// TIA Portal project "Poka Yoke Directa_V18" (V18)

(* hardware
DEVICE "S7-1200 station_1"  S7-1200 Station
   slot 0: "Rack_0"  S7-1200 Rack  Rack  V1.0
   slot 1: "PLC_1"  CPU 1215C DC/DC/Rly  6ES7 215-1HG40-0XB0  V4.6
DEVICE "GSD device_1"  GSD.Device.PN
   slot 0: "Rack"  Rack  V1.0
   slot 0: "smart-runner"  SmartRunner  310754  V3.1
      slot 0: "SmartRunner"  SmartRunner
      slot 1: "PN Interface"  PN Interface
         slot 1: "Port 1"  Port 1
         slot 2: "Port 2"  Port 2
   slot 1: "Head Address 1_1"  Head Address 1
      slot 0: "Head Address 1"  Head Address 1
*)

// ===== PLC "PLC_1"  CPU 1215C DC/DC/Rly =====

VAR_GLOBAL   // PLC tag table "PLC"
   "Pulsador Rojo Reset Desvio" AT %I0.0 : Bool;
   "No Match - RS482" AT %I0.1 : Bool;   // Sensor 2 - Mediante R482
   "Sensor Inductivo Soporte" AT %I0.2 : Bool;
   "Error" AT %I68.0 : Bool;
   "No Match - Profinet" AT %I68.1 : Bool;   // Sensor 1 - Profinet
   "Warning" AT %I68.2 : Bool;
   "Event" AT %I68.3 : Bool;
   "Status_addr" AT %I68.4 : Bool;
   "Status_addr 1" AT %I68.5 : Bool;
   "Result" AT %IB69 : Byte;
   "Counter" AT %IB70 : Byte;
   "Quality A" AT %IB71 : Byte;
   "Quality B" AT %IB72 : Byte;
   "Quality C" AT %IB73 : Byte;
   "Pos X" AT %IW74 : Int;
   "Pos Z" AT %IW76 : Int;
   "Checksum" AT %IB78 : Byte;
   "Rele Baliza" AT %Q0.3 : Bool;
   "Piloto Pulsador Rojo" AT %Q0.0 : Bool;
   "Rele bocina intermitente" AT %Q0.1 : Bool;
   "Trigger" AT %Q69.0 : Bool;
   "Teach" AT %Q71.0 : Bool;
   "Choose Profile" AT %QB73 : Byte;
   "Parada Gantry" AT %Q0.4 : Bool;
   "Piloto Error CPU" AT %Q0.5 : Bool;
   "Piloto OK" AT %Q0.2 : Bool;
   "Flanco Sensor Inductivo" AT %M0.2 : Bool;
   "Resultante" AT %MW10 : Int;
   "PF_Profinet" AT %MW2 : Hw_Io;
   "PF_LED" AT %MW4 : UInt;
   "System_Byte" AT %MB500 : Byte;
   "FirstScan" AT %M500.0 : Bool;
   "DiagStatusUpdate" AT %M500.1 : Bool;
   "AlwaysTRUE" AT %M500.2 : Bool;
   "AlwaysFALSE" AT %M500.3 : Bool;
   "Prueba" AT %M0.0 : Bool;
END_VAR

DATA_BLOCK "DataLogger_DB"   // DB9
{ S7_Optimized_Access := 'TRUE' }
VERSION : 0.1
// stored: InstanceOfName DataLogger
"DataLogger"
BEGIN
END_DATA_BLOCK

DATA_BLOCK "Control DataLogger"   // DB10
{ S7_Optimized_Access := 'TRUE' }
VERSION : 0.1
   VAR
      "Abrir Archivo" : Bool;
      "Escribir Archivo" : Bool;
      "Crear Archivo" : Bool;
      "Cerrar Archivo" : Bool;
      ID : DWord := 16#20;
   END_VAR
   VAR RETAIN
      "Name" : String;
   END_VAR
   VAR
      Data : Struct
         "Sensor 1" : Bool;
         "Sensor 2" : Bool;
         "Conexion Profinet" : Bool;
         "Quality A" : Int;
         "Quality B" : Int;
         "Quality C" : Int;
      END_STRUCT;
   END_VAR
BEGIN
END_DATA_BLOCK

// folder: 10_Sensor Doble

DATA_BLOCK "Status_LED"   // DB13
{ S7_Optimized_Access := 'TRUE' }
VERSION : 0.1
   VAR
      HW : Hw_Io := 50;
      LED : UInt := 2;
      "Return" : Int;
   END_VAR
BEGIN
END_DATA_BLOCK

// folder: FBs

DATA_BLOCK "SmartRunnner_Control_DB"   // DB8
{ S7_Optimized_Access := 'TRUE' }
VERSION : 0.1
// stored: InstanceOfName SmartRunnner_Control
"SmartRunnner_Control"
BEGIN
END_DATA_BLOCK

// folder: System blocks/Program resources

DATA_BLOCK "Temporizador TON Lectura de Datos"   // DB1
{ S7_Optimized_Access := 'TRUE' }
AUTHOR : Simatic
FAMILY : IEC
NAME : IEC_TMR
VERSION : 1.0
// stored: InstanceOfName IEC_TIMER
"IEC_TIMER"
BEGIN
END_DATA_BLOCK

DATA_BLOCK "Temporizador TON Pulsador Rojo"   // DB2
{ S7_Optimized_Access := 'TRUE' }
AUTHOR : Simatic
FAMILY : IEC
NAME : IEC_TMR
VERSION : 1.0
// stored: InstanceOfName IEC_TIMER
"IEC_TIMER"
BEGIN
END_DATA_BLOCK

DATA_BLOCK "Temporizador TP Pulsador Rojo"   // DB3
{ S7_Optimized_Access := 'TRUE' }
AUTHOR : Simatic
FAMILY : IEC
NAME : IEC_TMR
VERSION : 1.0
// stored: InstanceOfName IEC_TIMER
"IEC_TIMER"
BEGIN
END_DATA_BLOCK

DATA_BLOCK "Temporizador TP Reset"   // DB4
{ S7_Optimized_Access := 'TRUE' }
AUTHOR : Simatic
FAMILY : IEC
NAME : IEC_TMR
VERSION : 1.0
// stored: InstanceOfName IEC_TIMER
"IEC_TIMER"
BEGIN
END_DATA_BLOCK

DATA_BLOCK "Temporizador TON Reset"   // DB5
{ S7_Optimized_Access := 'TRUE' }
AUTHOR : Simatic
FAMILY : IEC
NAME : IEC_TMR
VERSION : 1.0
// stored: InstanceOfName IEC_TIMER
"IEC_TIMER"
BEGIN
END_DATA_BLOCK

DATA_BLOCK "TON_BOCINA"   // DB6
{ S7_Optimized_Access := 'TRUE' }
AUTHOR : Simatic
FAMILY : IEC
NAME : IEC_TMR
VERSION : 1.0
// stored: InstanceOfName IEC_TIMER
"IEC_TIMER"
BEGIN
END_DATA_BLOCK

DATA_BLOCK "TP_BOCINA"   // DB7
{ S7_Optimized_Access := 'TRUE' }
AUTHOR : Simatic
FAMILY : IEC
NAME : IEC_TMR
VERSION : 1.0
// stored: InstanceOfName IEC_TIMER
"IEC_TIMER"
BEGIN
END_DATA_BLOCK

DATA_BLOCK "TP Guardado"   // DB11
{ S7_Optimized_Access := 'TRUE' }
AUTHOR : Simatic
FAMILY : IEC
NAME : IEC_TMR
VERSION : 1.0
// stored: InstanceOfName IEC_TIMER
"IEC_TIMER"
BEGIN
END_DATA_BLOCK

DATA_BLOCK "Temporizador TON Giro Pieza"   // DB12
{ S7_Optimized_Access := 'TRUE' }
AUTHOR : Simatic
FAMILY : IEC
NAME : IEC_TMR
VERSION : 1.0
// stored: InstanceOfName IEC_TIMER
"IEC_TIMER"
BEGIN
END_DATA_BLOCK

DATA_BLOCK "TON Guardado"   // DB14
{ S7_Optimized_Access := 'TRUE' }
AUTHOR : Simatic
FAMILY : IEC
NAME : IEC_TMR
VERSION : 1.0
// stored: InstanceOfName IEC_TIMER
"IEC_TIMER"
BEGIN
END_DATA_BLOCK

DATA_BLOCK "Temporizador TP Lectura de Datos"   // DB25
{ S7_Optimized_Access := 'TRUE' }
AUTHOR : Simatic
FAMILY : IEC
NAME : IEC_TMR
VERSION : 1.0
// stored: InstanceOfName IEC_TIMER
"IEC_TIMER"
BEGIN
END_DATA_BLOCK

// folder: (top level)

FUNCTION_BLOCK "DataLogger"   // FB2, LAD
{ S7_Optimized_Access := 'TRUE' }
VERSION : 0.1
   VAR_INPUT
      LogCreate : Bool;
      LogOpen : Bool;
      LogWrite : Bool;
      LogClose : Bool;
      "Name" : String := 'Datalogger';
   END_VAR
   VAR_IN_OUT
      Data : Struct
         RS482 : Bool;
         Profinet : Bool;
         "Conexion Profinet" : Bool;
         "Quality A" : Int;
         "Quality B" : Int;
         "Quality C" : Int;
      END_STRUCT;
      ID : DWord := 16#20;
   END_VAR
   VAR
      Create : DataLogCreate;
      Header : String := 'RS482,Profinet,Conexion Profinet,Quality A, Quality B, Quality C';
      CreateDone : Bool;
      Write : DataLogWrite;
      WriteDone : Bool;
      OpenDone : Bool;
      Open : DataLogOpen;
      DataLogClose : DataLogClose;
   END_VAR
   VAR CONSTANT
      Records : UDInt := 20000;
      Format : UInt := 1;
      Timestamp : UInt := 4;
      Mode : UInt := 0;
   END_VAR
BEGIN

REGION Network 1
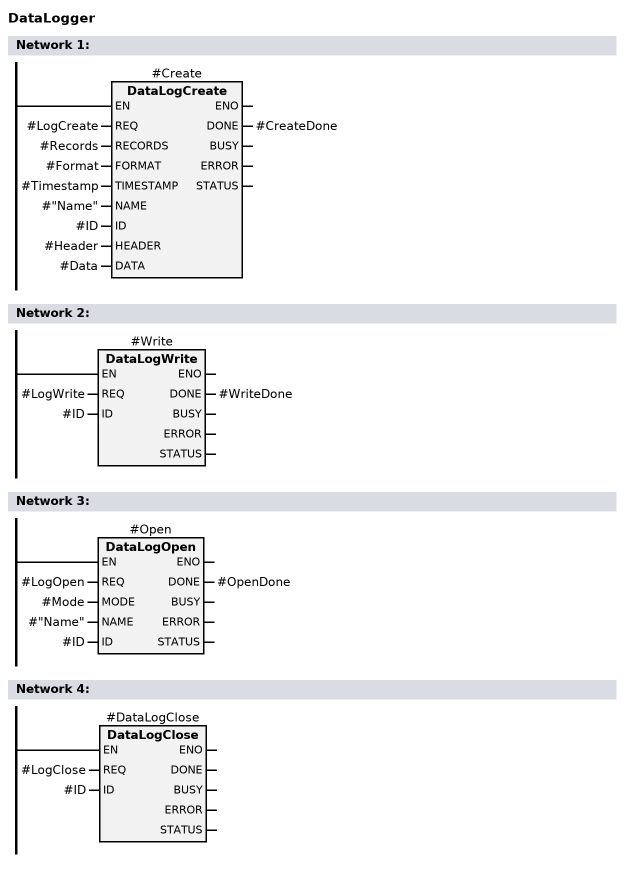
   #Create(REQ := #LogCreate,   // DataLogCreate
           RECORDS := #Records,
           FORMAT := #Format,
           TIMESTAMP := #Timestamp,
           "NAME" := #"Name",
           ID := #ID,
           HEADER := #Header,
           DATA := #Data,
           DONE => #CreateDone);
END_REGION

REGION Network 2
   #Write(REQ := #LogWrite, ID := #ID, DONE => #WriteDone);   // DataLogWrite
END_REGION

REGION Network 3
   #Open(REQ := #LogOpen, MODE := #Mode, "NAME" := #"Name", ID := #ID, DONE => #OpenDone);   // DataLogOpen
END_REGION

REGION Network 4
   #DataLogClose(REQ := #LogClose, ID := #ID);   // DataLogClose
END_REGION
END_FUNCTION_BLOCK

FUNCTION "Conversion Byte a Int" : Void   // FC2, LAD
{ S7_Optimized_Access := 'TRUE' }
VERSION : 0.1
BEGIN

REGION Network 1 (SCL)
   //comentario de prueba
   "Control DataLogger".Data."Quality A" :=  BYTE_TO_INT(IN :="Quality A");
   "Control DataLogger".Data."Quality B" := BYTE_TO_INT(IN := "Quality B");
   "Control DataLogger".Data."Quality C" := BYTE_TO_INT(IN := "Quality C");
END_REGION
END_FUNCTION

ORGANIZATION_BLOCK "Main"   // OB1, LAD, ProgramCycle
TITLE = "Main Program Sweep (Cycle)"
{ S7_Optimized_Access := 'TRUE' }
VERSION : 0.1
   VAR_INPUT
      Initial_Call : Bool;   // Initial call of this OB
      Remanence : Bool;   // =True, if remanent data are available
   END_VAR
BEGIN

REGION Network 1: Lectura del ambos sensores
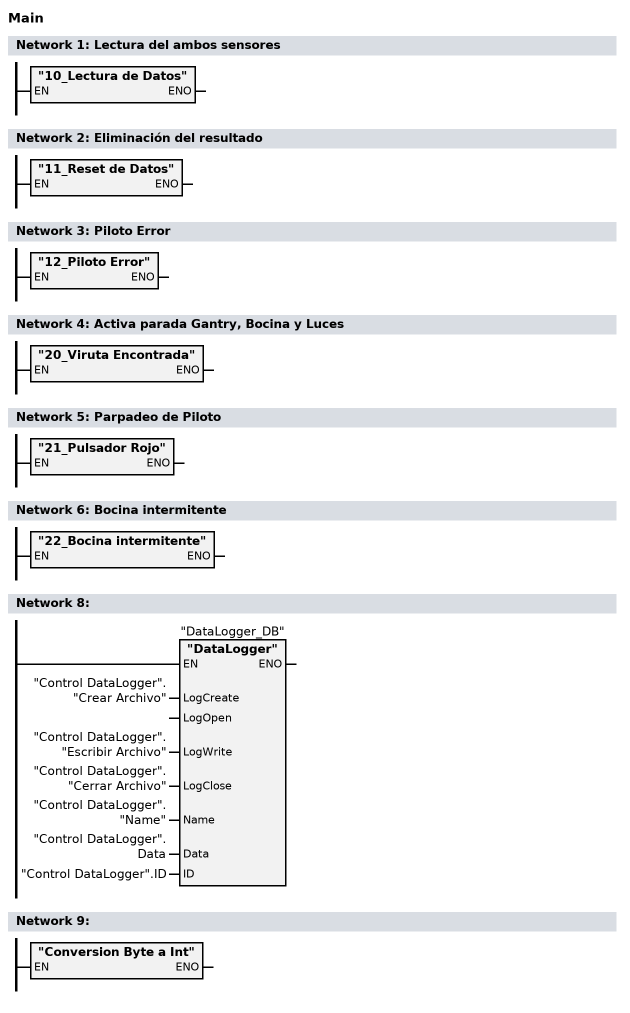
   RUNG wire#powerrail
      "10_Lectura de Datos"()
   END_RUNG
   // the same network as SCL:
   "10_Lectura de Datos"();
END_REGION

REGION Network 2: Eliminación del resultado
   RUNG wire#powerrail
      "11_Reset de Datos"()
   END_RUNG
   // the same network as SCL:
   "11_Reset de Datos"();
END_REGION

REGION Network 3: Piloto Error
   RUNG wire#powerrail
      "12_Piloto Error"()
   END_RUNG
   // the same network as SCL:
   "12_Piloto Error"();
END_REGION

REGION Network 4: Activa parada Gantry, Bocina y Luces
   RUNG wire#powerrail
      "20_Viruta Encontrada"()
   END_RUNG
   // the same network as SCL:
   "20_Viruta Encontrada"();
END_REGION

REGION Network 5: Parpadeo de Piloto
   RUNG wire#powerrail
      "21_Pulsador Rojo"()
   END_RUNG
   // the same network as SCL:
   "21_Pulsador Rojo"();
END_REGION

REGION Network 6: Bocina intermitente
   RUNG wire#powerrail
      "22_Bocina intermitente"()
   END_RUNG
   // the same network as SCL:
   "22_Bocina intermitente"();
END_REGION

REGION Network 7 (SCL)
   "Control DataLogger".Data."Sensor 1" := "No Match - RS482";
   "Control DataLogger".Data."Sensor 2" := "No Match - Profinet";
   "Control DataLogger".Data."Conexion Profinet" := "Piloto Error CPU";
END_REGION

REGION Network 8
   RUNG wire#powerrail
      "DataLogger_DB"(LogCreate := "Control DataLogger"."Crear Archivo", LogOpen :=, LogWrite := "Control DataLogger"."Escribir Archivo", LogClose := "Control DataLogger"."Cerrar Archivo", "Name" := "Control DataLogger"."Name", Data := "Control DataLogger".Data, ID := "Control DataLogger".ID)
   END_RUNG
   // the same network as SCL:
   "DataLogger_DB"(LogCreate := "Control DataLogger"."Crear Archivo",   // "DataLogger"
                   LogWrite := "Control DataLogger"."Escribir Archivo",
                   LogClose := "Control DataLogger"."Cerrar Archivo",
                   "Name" := "Control DataLogger"."Name",
                   Data := "Control DataLogger".Data,
                   ID := "Control DataLogger".ID);
END_REGION

REGION Network 9
   RUNG wire#powerrail
      "Conversion Byte a Int"()
   END_RUNG
   // the same network as SCL:
   "Conversion Byte a Int"();
END_REGION
END_ORGANIZATION_BLOCK

// folder: 10_Sensor Doble

FUNCTION "12_Piloto Error" : Void   // FC1, LAD
{ S7_Optimized_Access := 'TRUE' }
VERSION : 0.1
   VAR_TEMP
      PepperF_profinet : Hw_Io;
   END_VAR
BEGIN

REGION Network 1
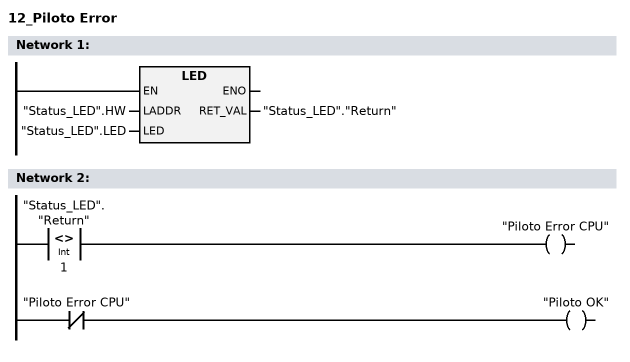
   "Status_LED"."Return" := LED(LADDR := "Status_LED".HW, LED := "Status_LED".LED);
END_REGION

REGION Network 2
   RUNG wire#powerrail
      { S7_Templates := "SrcType := Int" } NE_Contact(in1 := "Status_LED"."Return", in2 := 1)
      Coil( "Piloto Error CPU" )
   END_RUNG
   RUNG wire#powerrail
      I_Contact( "Piloto Error CPU" )
      Coil( "Piloto OK" )
   END_RUNG
   // the same network as SCL:
   "Piloto Error CPU" := "Status_LED"."Return" <> 1;
   "Piloto OK" := NOT "Piloto Error CPU";
END_REGION
END_FUNCTION

FUNCTION "10_Lectura de Datos" : Void   // FC20, LAD
{ S7_Optimized_Access := 'TRUE' }
VERSION : 0.1
   VAR_TEMP   // added for the SCL form of the ladder/FBD networks
      _w1 : Bool;
   END_VAR
BEGIN

REGION Network 1
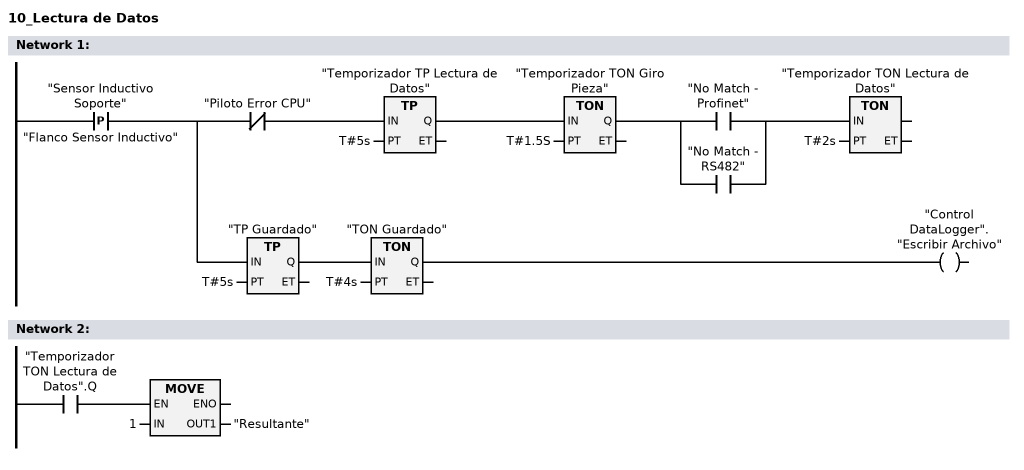
   #_w1 := "Sensor Inductivo Soporte" AND NOT "Flanco Sensor Inductivo";   // rising edge of "Sensor Inductivo Soporte"
   "Flanco Sensor Inductivo" := "Sensor Inductivo Soporte";
   "Temporizador TP Lectura de Datos".TP(IN := #_w1 AND NOT "Piloto Error CPU", PT := T#5s);
   "Temporizador TON Giro Pieza".TON(IN := "Temporizador TP Lectura de Datos".Q, PT := T#1.5S);
   "Temporizador TON Lectura de Datos".TON(IN := "Temporizador TON Giro Pieza".Q AND ("No Match - Profinet" OR "No Match - RS482"),
                           PT := T#2s);
   "TP Guardado".TP(IN := #_w1, PT := T#5s);
   "TON Guardado".TON(IN := "TP Guardado".Q, PT := T#4s);
   "Control DataLogger"."Escribir Archivo" := "TON Guardado".Q;
END_REGION

REGION Network 2
   RUNG wire#powerrail
      Contact( "Temporizador TON Lectura de Datos".Q )
      Move(in := 1, out1 => "Resultante")
   END_RUNG
   // the same network as SCL:
   IF "Temporizador TON Lectura de Datos".Q THEN "Resultante" := 1; END_IF;
END_REGION
END_FUNCTION

FUNCTION "11_Reset de Datos" : Void   // FC21, LAD
{ S7_Optimized_Access := 'TRUE' }
VERSION : 0.1
BEGIN

REGION Network 1
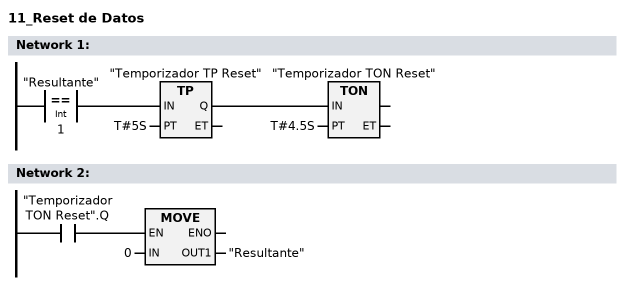
   "Temporizador TP Reset".TP(IN := "Resultante" = 1, PT := T#5S);
   "Temporizador TON Reset".TON(IN := "Temporizador TP Reset".Q, PT := T#4.5S);
END_REGION

REGION Network 2
   RUNG wire#powerrail
      Contact( "Temporizador TON Reset".Q )
      Move(in := 0, out1 => "Resultante")
   END_RUNG
   // the same network as SCL:
   IF "Temporizador TON Reset".Q THEN "Resultante" := 0; END_IF;
END_REGION
END_FUNCTION

// folder: 20_Movimientos

FUNCTION "20_Viruta Encontrada" : Void   // FC10, LAD
{ S7_Optimized_Access := 'TRUE' }
VERSION : 0.1
BEGIN

REGION Network 1
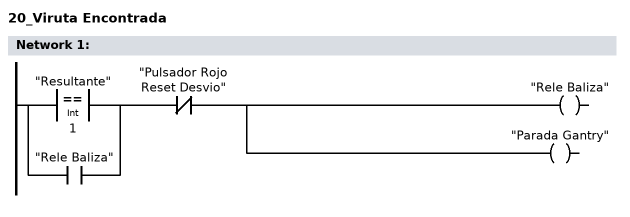
   RUNG wire#powerrail
      { S7_Templates := "SrcType := Int" } EQ_Contact(in1 := "Resultante", in2 := 1)
      wire#w1
      I_Contact( "Pulsador Rojo Reset Desvio" )
      wire#w2
      Coil( "Rele Baliza" )
   END_RUNG
   RUNG wire#powerrail
      Contact( "Rele Baliza" )
   END_RUNG wire#w1
   RUNG wire#w2
      Coil( "Parada Gantry" )
   END_RUNG
   // the same network as SCL:
   "Rele Baliza" := (("Resultante" = 1) OR "Rele Baliza") AND NOT "Pulsador Rojo Reset Desvio";
   "Parada Gantry" := "Rele Baliza";
END_REGION
END_FUNCTION

FUNCTION "21_Pulsador Rojo" : Void   // FC11, LAD
{ S7_Optimized_Access := 'TRUE' }
VERSION : 0.1
BEGIN

REGION Network 1
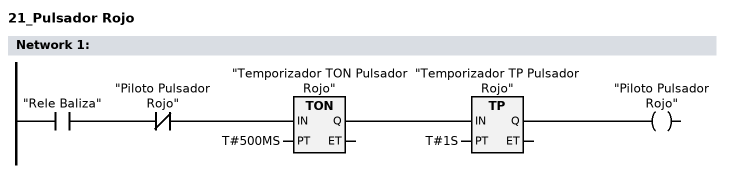
   "Temporizador TON Pulsador Rojo".TON(IN := "Rele Baliza" AND NOT "Piloto Pulsador Rojo", PT := T#500MS);
   "Temporizador TP Pulsador Rojo".TP(IN := "Temporizador TON Pulsador Rojo".Q, PT := T#1S);
   "Piloto Pulsador Rojo" := "Temporizador TP Pulsador Rojo".Q;
END_REGION
END_FUNCTION

FUNCTION "22_Bocina intermitente" : Void   // FC12, LAD
{ S7_Optimized_Access := 'TRUE' }
VERSION : 0.1
BEGIN

REGION Network 1
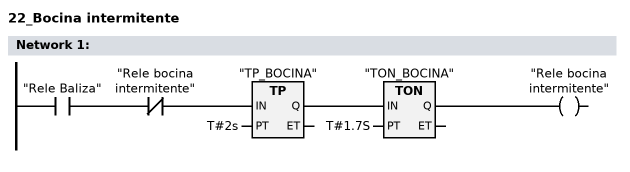
   "TP_BOCINA".TP(IN := "Rele Baliza" AND NOT "Rele bocina intermitente", PT := T#2s);
   "TON_BOCINA".TON(IN := "TP_BOCINA".Q, PT := T#1.7S);
   "Rele bocina intermitente" := "TON_BOCINA".Q;
END_REGION
END_FUNCTION

// folder: FBs

FUNCTION_BLOCK "SmartRunnner_Control"   // FB1, SCL
{ S7_Optimized_Access := 'TRUE' }
VERSION : 0.1
   VAR_INPUT
      REQ : Bool;
      HEAD_ADDR : Hw_Io;
      TRIGGER : Bool;
      TEACH : Bool;
      CHOOSE_PROFILE : Bool;
      PROFILE_NUMBER : USInt;
   END_VAR
   VAR_OUTPUT
      BUSY : Bool;
      DONE : Bool;
      TEACH_SET : Bool;
      TEACH_OK : Bool;
      ERROR : Bool;
      ERROR_ID : Byte;
      MATCH : Bool;
      NO_MATCH : Bool;
      PROFILE_NO : USInt;
      "COUNTER" : Byte;
      QUALITY_GOOD : USInt;
      QUALITY_VARIATION : USInt;
      QUALITY_OUTLIERS : USInt;
      X_OFFSET : Int;
      Z_OFFSET : Int;
   END_VAR
   VAR
      TRANSMIT : Struct
         Reserved : Byte;
         Trigger : Byte;
         Reserved_1 : Byte;
         Teach : Byte;
         Reserved_2 : Byte;
         Profile : Byte;
      END_STRUCT;
      RESPONSE : Struct
         Status : Byte;
         Result : Byte;
         "Counter" : Byte;
         Quality_Good : Byte;
         Quality_Var : Byte;
         Quality_Out : Byte;
         PosX_High : Byte;
         PosX_Low : Byte;
         PosZ_High : Byte;
         PosZ_Low : Byte;
         Checksum : Byte;
         Reserved : Byte;
         Reserved_1 : Byte;
         Reserved_2 : Byte;
         Reserved_3 : Byte;
         Handshake : Byte;
         TEACH_Status : Byte;
         TEACH_Result : Byte;
         TEACH_Counter : Byte;
         TEACH_QualityA : Byte;
         TEACH_QualityB : Byte;
         TEACH_QualityC : Byte;
         TEACH_QualityD : Byte;
         TEACH_Checksum : Byte;
      END_STRUCT;
      R_TRIG_TRIGGER : R_TRIG;
      Processing : Bool;
      Failure : Bool;
      RetVal_SFC14 : Int;
      RetVal_SFC15 : Int;
      PreviousCtr : Byte;
      PreviousTeachCtr : Byte;
      Trigger_Active : Bool;
      Teach_Active : Bool;
      Profile_Active : Bool;
      IEC_Timer_Watchdog : TON_TIME;
      myXpos : Word;
      myXposBits AT myXpos : Array[0..15] of Bool;
      "my Zpos" : Word;
      myZposBits AT "my Zpos" : Array[0..15] of Bool;
      IEC_Timer_Delay : TON_TIME;
   END_VAR
BEGIN
   (* 
   Function block to trigger, teach and choose profiles for SmartRunner (VLX-F231-B17).

   Date: 23.01.2020
   Version: 1.0.2 
   Features:
   - handshake bits evaluation added
   - minor adjustments and bug fixes in source code

   Date: 01.08.2019
   Version: 1.0 
   Features:
   - software trigger added
   - utilize process data after software trigger
   - teach profiles added
   - choose profiles added
   - sanity check for input variables 
   *)

   REGION Retrieve SmartRunnner data and allocate outputs
   (* Read from BUS *)       
   #RetVal_SFC14 := DPRD_DAT(LADDR := #HEAD_ADDR, RECORD => #RESPONSE);

   IF #RetVal_SFC14 = 0 THEN

       (* Match / No Match *)
       IF (#RESPONSE.Status AND 16#02) = 16#02 THEN
           #NO_MATCH := TRUE;
           #MATCH := FALSE;
       ELSE
           #NO_MATCH := FALSE;
           #MATCH := TRUE;
       END_IF;

       (* Error *)
       IF (#RESPONSE.Status AND 16#1) = 16#1 THEN
           #ERROR := TRUE;
           #ERROR_ID := 2;
       END_IF;

       (* Profile number *)
       #PROFILE_NO := #RESPONSE.Result;

       (* Counter *)
       #COUNTER := #RESPONSE.Counter;

       (* Qualities *)
       #QUALITY_GOOD := #RESPONSE.Quality_Good;
       #QUALITY_VARIATION := #RESPONSE.Quality_Var;
       #QUALITY_OUTLIERS := #RESPONSE.Quality_Out;


       (* X Offset *)
       IF (#RESPONSE.PosX_High AND 16#01) = 16#01 THEN
           #myXpos := SHR(IN := BYTE_TO_WORD(#RESPONSE.PosX_High), N := 1);
           #myXpos := SHL(IN := #myXpos, N := 8) OR BYTE_TO_WORD((#RESPONSE.PosX_Low OR 16#80));  (* Concatenate High + Low Byte of X_Pos *)
           IF #myXposBits[13] THEN (* Check for negativ number and convert *)
               #myXpos := (((NOT #myXpos) AND 16#3FFF) + 1);
               #X_OFFSET := WORD_TO_INT(#myXpos) * (-1);
           END_IF;
       ELSE
           #myXpos := SHR(IN := BYTE_TO_WORD(#RESPONSE.PosX_High), N := 1);
           #myXpos := SHL(IN := #myXpos, N := 8) OR BYTE_TO_WORD(#RESPONSE.PosX_Low);
           #X_OFFSET := WORD_TO_INT(#myXpos);
       END_IF;

       (* Z Offset *)
       IF (#RESPONSE.PosZ_High AND 16#01) = 16#01 THEN
           #"my Zpos" := SHR(IN := BYTE_TO_WORD(#RESPONSE.PosZ_High), N := 1);
           #"my Zpos" := SHL(IN := #"my Zpos", N := 8) OR BYTE_TO_WORD((#RESPONSE.PosZ_Low OR 16#80));
           IF #myZposBits[13] THEN
               #"my Zpos" := (((NOT #"my Zpos") AND 16#3FFF) + 1);
               #Z_OFFSET := WORD_TO_INT(#"my Zpos") * (-1);
           END_IF;
       ELSE
           #"my Zpos" := SHR(IN := BYTE_TO_WORD(#RESPONSE.PosZ_High), N := 1);
           #"my Zpos" := SHL(IN := #"my Zpos", N := 8) OR BYTE_TO_WORD(#RESPONSE.PosZ_Low);
           #Z_OFFSET := WORD_TO_INT(#"my Zpos");
       END_IF;

   ELSE
       #ERROR := TRUE;
       #ERROR_ID := 1;
   END_IF;
   END_REGION

   REGION Multiple input check
   IF #TRIGGER AND (#TEACH OR #CHOOSE_PROFILE) OR
           #TEACH AND (#TRIGGER OR #CHOOSE_PROFILE) OR
               #CHOOSE_PROFILE AND (#TRIGGER OR #TEACH) THEN
       #ERROR := TRUE;
       #ERROR_ID := 3; (* Multiple inputs *)
       RETURN; (* Do nothing and return *)
   END_IF;
   END_REGION

   REGION TRIGGER, TEACH, PROFILE
   #R_TRIG_TRIGGER(CLK := #REQ);

   IF #R_TRIG_TRIGGER.Q AND NOT #Processing THEN
       #BUSY := TRUE;
       #DONE := FALSE;
       #ERROR := FALSE;
       #Failure := FALSE;
       #ERROR_ID := 16#00;
       #Processing := TRUE;

       (* Assemble bits for output command *)
       IF #TRIGGER THEN
           #TRANSMIT.Trigger := 16#01;
           #Trigger_Active := TRUE;
       ELSIF #TEACH THEN
           #TRANSMIT.Teach := 16#01;
           #Teach_Active := TRUE;
       ELSIF #CHOOSE_PROFILE THEN
           #TRANSMIT.Profile := #PROFILE_NUMBER;
           #Profile_Active := TRUE;
       END_IF;

       (* Write output *)
       #RetVal_SFC15 := DPWR_DAT(LADDR := #HEAD_ADDR, RECORD := #TRANSMIT);
   END_IF;

   (* Evaluate new response *)
   IF #RetVal_SFC15 = 0 AND #RetVal_SFC14 = 0 AND #Processing THEN
       (* Reset outputs *)        
       IF #RESPONSE.Handshake.%X0 THEN (* Softwaretrigger ACK *)
           #TRANSMIT.Trigger := 16#00;
           (* Write output *)
           #RetVal_SFC15 := DPWR_DAT(LADDR := #HEAD_ADDR, RECORD := #TRANSMIT);
       ELSIF #RESPONSE.Handshake.%X1 THEN (* Update Profile ACK *)
           #TRANSMIT.Profile := 16#00;
           #Profile_Active := FALSE;
           #Processing := FALSE;
           (* Write output *)
           #RetVal_SFC15 := DPWR_DAT(LADDR := #HEAD_ADDR, RECORD := #TRANSMIT);
       ELSIF #RESPONSE.Handshake.%X2 THEN (* Teach ACK *)
           #TRANSMIT.Teach := 16#00;
           #TEACH_SET := TRUE;
           #TEACH_OK := FALSE;
           #Processing := FALSE;
           (* Write output *)
           #RetVal_SFC15 := DPWR_DAT(LADDR := #HEAD_ADDR, RECORD := #TRANSMIT);
       END_IF;

       (* Trigger Response available *)
       IF (#PreviousCtr <> #RESPONSE.Counter) AND #Trigger_Active THEN

           #PreviousCtr := #RESPONSE.Counter;
           #Trigger_Active := FALSE;

           (* Operation finished *)
           #Processing := FALSE;

       (* Response for TEACH command after TRIGGER *)
       ELSIF (#RESPONSE.TEACH_Counter <> #PreviousTeachCtr) AND #Teach_Active AND #Trigger_Active THEN

           #PreviousTeachCtr := #RESPONSE.TEACH_Counter;
           #Teach_Active := FALSE;
           #Trigger_Active := FALSE;

           IF #RESPONSE.TEACH_QualityA <> 16#00 THEN (* TEACH okay *)
               #TEACH_OK := TRUE;
               #TEACH_SET := FALSE;
           ELSE                                    (* TEACH failed *)
               #TEACH_OK := FALSE;
               #TEACH_SET := FALSE;
               #Failure := TRUE;
               #ERROR_ID := 16#FE;
           END_IF;

           #Processing := FALSE;
       END_IF;
   END_IF;
   END_REGION

   REGION Watchdog
   #IEC_Timer_Watchdog(IN := #Processing,
                       PT := T#10s);
   (* Reset everything *)
   IF #IEC_Timer_Watchdog.Q THEN
       #Processing := FALSE;
       #Failure := TRUE;
       #ERROR_ID := 1;
   END_IF;
   END_REGION

   REGION Failure and output handling    
   (* Process finished and all Handshake bits in FALSE state *)
   IF NOT #Processing AND #RESPONSE.Handshake = 16#00 THEN
       #BUSY := FALSE;
       #DONE := TRUE;
       IF #Failure THEN  (* Reset outputs *)
           #TRANSMIT.Trigger := 16#00;
           #TRANSMIT.Teach := 16#00;
           #TRANSMIT.Profile := 16#00;
           #ERROR := TRUE;

           #RetVal_SFC15 := DPWR_DAT(LADDR := #HEAD_ADDR, RECORD := #TRANSMIT);
       END_IF;
   END_IF;
   END_REGION
END_FUNCTION_BLOCK